PROGRAM PRG_IN_VACUUM_MOTION
VAR

	(* Axis X1 *)
	{attribute 'TcLinkToOSO' := '
		.stDS402Drive.nModeOfOperationNC      := <0,8,0>TINC^NC-Task 1^Axes^M13_DREAM_SLIT_MMT_X1^Drive^Outputs^Out^nCtrl5;
		.stDS402Drive.nDS402DriveControlNC.0  := <0,8,0>TINC^NC-Task 1^Axes^M13_DREAM_SLIT_MMT_X1^Drive^Outputs^Out^nCtrl1;
		.stDS402Drive.nDS402DriveControlNC.1  := <8,8,0>TINC^NC-Task 1^Axes^M13_DREAM_SLIT_MMT_X1^Drive^Outputs^Out^nCtrl2;
	'}
	{attribute 'TcLinkTo' := '
		.stDS402Drive.nSlaveAddr              := TIID^Device 1 (EtherCAT)^TMO-DREAM-SMARACT-04^InfoData^AdsAddr^port;
		.stDS402Drive.stDS402DriveStatus      := TIID^Device 1 (EtherCAT)^TMO-DREAM-SMARACT-04^DREAM:SLIT:MMT:X1^mode/status/pos/fError TxPDO^Status Word;
		.stDS402Drive.nFollowingError         := TIID^Device 1 (EtherCAT)^TMO-DREAM-SMARACT-04^DREAM:SLIT:MMT:X1^mode/status/pos/fError TxPDO^Following Error Actual Value;
		.stDS402Drive.nModeOfOperation        := TIID^Device 1 (EtherCAT)^TMO-DREAM-SMARACT-04^DREAM:SLIT:MMT:X1^ctl/mode/pos RxPDO^Modes of Operation;
		.stDS402Drive.nModeOfOperationDisplay := TIID^Device 1 (EtherCAT)^TMO-DREAM-SMARACT-04^DREAM:SLIT:MMT:X1^mode/status/pos/fError TxPDO^Modes of Operation Display;
		.stDS402Drive.nDS402DriveControl      := TIID^Device 1 (EtherCAT)^TMO-DREAM-SMARACT-04^DREAM:SLIT:MMT:X1^ctl/mode/pos RxPDO^Control Word;
	'}
	fb_SLIT_X1 : FB_MotionStageMCS2(stPiezoStage:=Main.M13 , eModule:=E_Module.CHAN2);
	
	(* Axis X2 *)
	{attribute 'TcLinkToOSO' := '
		.stDS402Drive.nModeOfOperationNC      := <0,8,0>TINC^NC-Task 1^Axes^M14_DREAM_SLIT_MMT_X2^Drive^Outputs^Out^nCtrl5;
		.stDS402Drive.nDS402DriveControlNC.0  := <0,8,0>TINC^NC-Task 1^Axes^M14_DREAM_SLIT_MMT_X2^Drive^Outputs^Out^nCtrl1;
		.stDS402Drive.nDS402DriveControlNC.1  := <8,8,0>TINC^NC-Task 1^Axes^M14_DREAM_SLIT_MMT_X2^Drive^Outputs^Out^nCtrl2;
	'}
	{attribute 'TcLinkTo' := '
		.stDS402Drive.nSlaveAddr              := TIID^Device 1 (EtherCAT)^TMO-DREAM-SMARACT-04^InfoData^AdsAddr^port;
		.stDS402Drive.stDS402DriveStatus      := TIID^Device 1 (EtherCAT)^TMO-DREAM-SMARACT-04^DREAM:SLIT:MMT:X2^mode/status/pos/fError TxPDO^Status Word;
		.stDS402Drive.nFollowingError         := TIID^Device 1 (EtherCAT)^TMO-DREAM-SMARACT-04^DREAM:SLIT:MMT:X2^mode/status/pos/fError TxPDO^Following Error Actual Value;
		.stDS402Drive.nModeOfOperation        := TIID^Device 1 (EtherCAT)^TMO-DREAM-SMARACT-04^DREAM:SLIT:MMT:X2^ctl/mode/pos RxPDO^Modes of Operation;
		.stDS402Drive.nModeOfOperationDisplay := TIID^Device 1 (EtherCAT)^TMO-DREAM-SMARACT-04^DREAM:SLIT:MMT:X2^mode/status/pos/fError TxPDO^Modes of Operation Display;
		.stDS402Drive.nDS402DriveControl      := TIID^Device 1 (EtherCAT)^TMO-DREAM-SMARACT-04^DREAM:SLIT:MMT:X2^ctl/mode/pos RxPDO^Control Word;
	'}
	fb_SLIT_X2 : FB_MotionStageMCS2(stPiezoStage:=Main.M14, eModule:=E_Module.CHAN3);
	
	(* Axis Y1 *)
	{attribute 'TcLinkToOSO' := '
		.stDS402Drive.nModeOfOperationNC      := <0,8,0>TINC^NC-Task 1^Axes^M15_DREAM_SLIT_MMT_Y1^Drive^Outputs^Out^nCtrl5;
		.stDS402Drive.nDS402DriveControlNC.0  := <0,8,0>TINC^NC-Task 1^Axes^M15_DREAM_SLIT_MMT_Y1^Drive^Outputs^Out^nCtrl1;
		.stDS402Drive.nDS402DriveControlNC.1  := <8,8,0>TINC^NC-Task 1^Axes^M15_DREAM_SLIT_MMT_Y1^Drive^Outputs^Out^nCtrl2;
	'}
	{attribute 'TcLinkTo' := '
		.stDS402Drive.nSlaveAddr              := TIID^Device 1 (EtherCAT)^TMO-DREAM-SMARACT-05^InfoData^AdsAddr^port;
		.stDS402Drive.stDS402DriveStatus      := TIID^Device 1 (EtherCAT)^TMO-DREAM-SMARACT-05^DREAM:SLIT:MMT:Y1^mode/status/pos/fError TxPDO^Status Word;
		.stDS402Drive.nFollowingError         := TIID^Device 1 (EtherCAT)^TMO-DREAM-SMARACT-05^DREAM:SLIT:MMT:Y1^mode/status/pos/fError TxPDO^Following Error Actual Value;
		.stDS402Drive.nModeOfOperation        := TIID^Device 1 (EtherCAT)^TMO-DREAM-SMARACT-05^DREAM:SLIT:MMT:Y1^ctl/mode/pos RxPDO^Modes of Operation;
		.stDS402Drive.nModeOfOperationDisplay := TIID^Device 1 (EtherCAT)^TMO-DREAM-SMARACT-05^DREAM:SLIT:MMT:Y1^mode/status/pos/fError TxPDO^Modes of Operation Display;
		.stDS402Drive.nDS402DriveControl      := TIID^Device 1 (EtherCAT)^TMO-DREAM-SMARACT-05^DREAM:SLIT:MMT:Y1^ctl/mode/pos RxPDO^Control Word;
	'}
	fb_SLIT_Y1 : FB_MotionStageMCS2(stPiezoStage:=Main.M15, eModule:=E_Module.CHAN1);
	
	(* Axis Y2 *)
	{attribute 'TcLinkToOSO' := '
		.stDS402Drive.nModeOfOperationNC      := <0,8,0>TINC^NC-Task 1^Axes^M16_DREAM_SLIT_MMT_Y2^Drive^Outputs^Out^nCtrl5;
		.stDS402Drive.nDS402DriveControlNC.0  := <0,8,0>TINC^NC-Task 1^Axes^M16_DREAM_SLIT_MMT_Y2^Drive^Outputs^Out^nCtrl1;
		.stDS402Drive.nDS402DriveControlNC.1  := <8,8,0>TINC^NC-Task 1^Axes^M16_DREAM_SLIT_MMT_Y2^Drive^Outputs^Out^nCtrl2;
	'}
	{attribute 'TcLinkTo' := '
		.stDS402Drive.nSlaveAddr              := TIID^Device 1 (EtherCAT)^TMO-DREAM-SMARACT-05^InfoData^AdsAddr^port;
		.stDS402Drive.stDS402DriveStatus      := TIID^Device 1 (EtherCAT)^TMO-DREAM-SMARACT-05^DREAM:SLIT:MMT:Y2^mode/status/pos/fError TxPDO^Status Word;
		.stDS402Drive.nFollowingError         := TIID^Device 1 (EtherCAT)^TMO-DREAM-SMARACT-05^DREAM:SLIT:MMT:Y2^mode/status/pos/fError TxPDO^Following Error Actual Value;
		.stDS402Drive.nModeOfOperation        := TIID^Device 1 (EtherCAT)^TMO-DREAM-SMARACT-05^DREAM:SLIT:MMT:Y2^ctl/mode/pos RxPDO^Modes of Operation;
		.stDS402Drive.nModeOfOperationDisplay := TIID^Device 1 (EtherCAT)^TMO-DREAM-SMARACT-05^DREAM:SLIT:MMT:Y2^mode/status/pos/fError TxPDO^Modes of Operation Display;
		.stDS402Drive.nDS402DriveControl      := TIID^Device 1 (EtherCAT)^TMO-DREAM-SMARACT-05^DREAM:SLIT:MMT:Y2^ctl/mode/pos RxPDO^Control Word;
	'}
	fb_SLIT_Y2 : FB_MotionStageMCS2(stPiezoStage:=Main.M16, eModule:=E_Module.CHAN2);
END_VAR

END_PROGRAM

(* stored: Version 1.1.0.1
   POU PRG_IN_VACUUM_MOTION: Id {cda8fdc4-ad80-409c-9b3b-55790280c462}, SpecialFunc None *)
